// TIA Portal V20 export
TYPE "OPC_SegmentStatus"
// stored: Namespace ProductionLine
   STRUCT
      Segment : Struct
         FlowRackLoop : Int;
         FlowRackWorkplaceLeft : Int;
         FlowRackWorkplaceRight : Int;
         FragileLoop : Int;
      END_STRUCT;
   END_STRUCT;
END_TYPE
